FUNCTION_BLOCK BUTTONdriver
VAR_INPUT
	buttonChannel : UINT := 1;
END_VAR
VAR_OUTPUT
END_VAR
VAR
	ch1 AT %I* : BOOL;
	ch2 AT %I* : BOOL;
	ch3 AT %I* : BOOL;
	ch4 AT %I* : BOOL;
	ch5 AT %I* : BOOL;
	ch6 AT %I* : BOOL;
	ch7 AT %I* : BOOL;
	ch8 AT %I* : BOOL;
	
	tmr1 : TON;
	currentValue : BOOL := FALSE;
	executed : BOOL := FALSE;
	
	state : ButtonType := ButtonType.notPressed;
END_VAR

CASE buttonChannel OF
	1:
		currentValue := ch1;
	2:
		currentValue := ch2;
	3:
		currentValue := ch3;
	4:
		currentValue := ch4;
	5:
		currentValue := ch5;
	6:
		currentValue := ch6;
	7:
		currentValue := ch7;
	8:
		currentValue := ch8;
END_CASE

IF currentValue AND NOT executed THEN
	tmr1(IN := TRUE, PT := T#10S);
	executed := TRUE;
ELSIF executed AND NOT currentValue AND (tmr1.ET < T#2S) THEN
	//momentary press
	tmr1(IN := FALSE);
	executed := FALSE;
	state := buttonType.pressed;
ELSIF executed AND NOT currentValue AND (tmr1.ET > T#2S) AND (tmr1.ET < T#5S) THEN
	//2S press
	tmr1(IN := FALSE);
	executed := FALSE;
	state := buttonType.hold2s;
ELSIF executed AND NOT currentValue AND (tmr1.ET > T#5S) THEN
	//5S press
	tmr1(IN := FALSE);
	executed := FALSE;
	state := buttonType.hold5s;
ELSIF executed AND tmr1.Q THEN
	//longer than 10S
	tmr1(IN := FALSE);
	executed := FALSE;
	state := buttonType.hold5s;
END_IF
tmr1();

METHOD getValue : BOOL
VAR_INPUT
END_VAR
VAR_OUTPUT
	stateOut : ButtonType;
END_VAR
stateOut := state;
state := ButtonType.notPressed;
getValue := TRUE;
END_METHOD

END_FUNCTION_BLOCK

(* stored: Version 1.1.0.1, ProductVersion 3.1.4022.18
   POU BUTTONdriver: Id {ef721045-7985-4393-8e0d-8008f95e668b}, SpecialFunc None
   Method getValue: Id {1fbeb37e-6e19-43b4-920d-be92c6c5c331} *)
